FUNCTION_BLOCK FB_Feeder EXTENDS FB_Conveyor
VAR_INPUT
    // Follower is ready to receive part
    bReleasePartTransfer: BOOL;
    // Part is at conveyor exit
    bPartAtExit: BOOL;
END_VAR
VAR_OUTPUT
    // Enable part emitter
    bEmitter: BOOL;
END_VAR
VAR
    // Enable processing of parts
    bEnable: BOOL;
    // Timer for maximum part moving time on conveyor
    fbMaxMovingTime: TON;
    // Current state of feeder
    eStateFeeder: (F_IDLE, F_MOVE_PART, F_WAIT_FOR_FOLLOWER, F_TRANSFER_TO_FOLLOWER, F_EMPTY_CONVEYOR, F_LOCKOUT);
END_VAR

SUPER^();
fbMaxMovingTime();

CASE eStateFeeder OF
    F_IDLE:
        SUPER^.Stop(bRunOut := FALSE);
        IF bEnable THEN
            bEmitter := TRUE;
            eStateFeeder := F_MOVE_PART;
        END_IF

    F_MOVE_PART:
        SUPER^.Start();
        fbMaxMovingTime.IN := TRUE;
        IF MovePartMonitor() THEN
            fbMaxMovingTime.IN := FALSE;
        ELSIF fbMaxMovingTime.Q THEN
            // Throw error message: Part moving timeout
            bEmitter := FALSE;
            eStateFeeder := F_IDLE;
        END_IF

    F_WAIT_FOR_FOLLOWER:
        SUPER^.Stop(bRunOut := FALSE);
        IF NOT bPartAtExit THEN
            // Throw message: Part was manual removed
            bEmitter := FALSE;
            eStateFeeder := F_IDLE;
        END_IF
        IF bReleasePartTransfer THEN
            eStateFeeder := F_TRANSFER_TO_FOLLOWER;
        END_IF

    F_TRANSFER_TO_FOLLOWER:
        SUPER^.Start();
        IF NOT bPartAtExit AND NOT bEnable THEN
            eStateFeeder := F_EMPTY_CONVEYOR;
        ELSIF NOT bPartAtExit THEN
            eStateFeeder := F_MOVE_PART;
        END_IF

    F_EMPTY_CONVEYOR:
        bEmitter := FALSE;
        fbMaxMovingTime.IN := TRUE;
        IF MovePartMonitor() THEN
            fbMaxMovingTime.IN := FALSE;
        END_IF
        IF fbMaxMovingTime.Q THEN
            fbMaxMovingTime.IN := FALSE;
            eStateFeeder := F_IDLE;
        END_IF
END_CASE

// Unset enable
bEnable := FALSE;

// Enable processing of parts
METHOD Enable: BOOL
VAR_INPUT
END_VAR
bEnable := TRUE;
END_METHOD

// Return TRUE if part reach conveyor exit and state machine will go to next step
METHOD PRIVATE MovePartMonitor: BOOL
VAR_INPUT
END_VAR
IF bPartAtExit AND bReleasePartTransfer THEN
    eStateFeeder := F_TRANSFER_TO_FOLLOWER;
ELSIF bPartAtExit THEN
    eStateFeeder := F_WAIT_FOR_FOLLOWER;
ELSE
    MovePartMonitor := FALSE;
    RETURN;
END_IF

MovePartMonitor := TRUE;
END_METHOD

// Maximum duration for part to reach exit of conveyor
{attribute 'monitoring' := 'call'}
PROPERTY PUBLIC tMaxMovingTime : TIME
GET
tMaxMovingTime := fbMaxMovingTime.PT;
END_GET
SET
fbMaxMovingTime.PT := tMaxMovingTime;
END_SET
END_PROPERTY

END_FUNCTION_BLOCK

(* stored: Version 1.1.0.1
   POU FB_Feeder: Id {c5d8e8bc-afa3-42ac-9bb3-50daf9da39ed}, SpecialFunc None
   Method Enable: Id {5968398c-874e-4b04-a814-7d741cce27ab}
   Method MovePartMonitor: Id {c7305287-8257-4d92-8802-940a28b7e430}
   Property tMaxMovingTime: Id {29a45c02-ab1e-4262-8ddc-dfbb68084338}
   Get Get: Id {4a60306e-e9b7-4682-8cbb-3a15601b517d}
   Set Set: Id {ec94b853-c8d5-4b26-9137-79b8d1d43967} *)
